// TIA Portal V20 export
FUNCTION_BLOCK "FB_HMI_PLC_Pos"   // FB80, SCL
{ S7_Optimized_Access := 'TRUE' }
// stored: MemoryReserve 100, SetENOAutomatically false
   VAR_INPUT
      "HMI_Change Enable" : Bool;
   END_VAR
   VAR_IN_OUT
      ioPLC_State : Bool;
      ioHMI_State : Bool;
   END_VAR
   VAR
      PLC_StateMemo : Bool;
      HMI_StateMemo : Bool;
   END_VAR
BEGIN
   REGION Description header 
       //==================================================================================
       // POSALUX Swiss SA / (C) Copyright 2026
       //----------------------------------------------------------------------------------
       // Title: FB_HMI_PLC_Pos
       // Comment/Function: 
       // Author: Fabien WALDT
       // Engineering: TIA Portal v20
       //----------------------------------------------------------------------------------
       // Change log table:
       // Version  | Date     | Expert in charge | Changes applied
       // ---------|----------|------------------|-----------------------------------------
       // 00.00.01 | 20260521 | WFA              | First released version
       // =================================================================================
   END_REGION

   REGION Update Values
       IF #ioPLC_State <> #PLC_StateMemo OR NOT #"HMI_Change Enable" THEN
           #ioHMI_State := #ioPLC_State;
           #HMI_StateMemo := #ioPLC_State;
           #PLC_StateMemo := #ioPLC_State;
       ELSIF (#ioHMI_State <> #HMI_StateMemo) AND #"HMI_Change Enable" THEN
           #ioPLC_State := #ioHMI_State;
           #PLC_StateMemo := #ioHMI_State;
           #HMI_StateMemo := #ioHMI_State;
       END_IF;

   END_REGION
END_FUNCTION_BLOCK
